TYPE tchmi_framework_definitions_XtsMoverList : ARRAY[0..1] OF tchmi_framework_definitions_XtsMoverListItem;
END_TYPE

(* stored: Version 1.1.0.1, ProductVersion 3.1.4024.12
   DUT tchmi_framework_definitions_XtsMoverList: Id {41cbddb9-4d90-453b-b2f3-e4b9a9c050d0} *)
